TYPE ST_ORCA_ProductInfo :
STRUCT

	OutersPerRow 			: STRING(255);
	RowsPerCase	 		: STRING(255);


END_STRUCT
END_TYPE

(* stored: Version 1.1.0.1, ProductVersion 3.1.4024.15
   DUT ST_ORCA_ProductInfo: Id {04ca6183-b8ba-43b0-b000-03ec9e1e9d07} *)
